{attribute 'GeneratedUsingTerminal: EL6692-0002-0016'}
{attribute addProperty BoxType "EL6692-0002-0016"}
{attribute addProperty Id "SYNC_InputsAT %I*SYNC_Inputs_462ED3216IO_InputsEMPTY_STRUCTURE0IO_OutputsEMPTY_STRUCTURE0WcStateAT %I*WcState_9091E0EB2InfoDataAT %I*InfoData_41C547A32"}
{attribute addProperty CRC "3426393028"}
{attribute addProperty Size "10"}
TYPE EL6692_CC3A9BC4 EXTENDS EtcSlaveTerminalBase_947E5A46 :
STRUCT
	{attribute addProperty Name "SYNC_Inputs"}
	SYNC_Inputs : SYNC_Inputs_462ED321;
	{attribute addProperty Name "IO_Inputs"}
	IO_Inputs : EMPTY_STRUCTURE;
	{attribute addProperty Name "IO_Outputs"}
	IO_Outputs : EMPTY_STRUCTURE;
	{attribute addProperty Name "WcState"}
	WcState : WcState_9091E0EB;
	{attribute addProperty Name "InfoData"}
	InfoData : InfoData_41C547A3;
END_STRUCT
END_TYPE

(* stored: Version 1.2.0.0, ProductVersion 3.1.4024.9
   DUT EL6692_CC3A9BC4: Id {f7644964-daed-4601-8845-13f02cdf50cd} *)
